FUNCTION_BLOCK FB_Observer_LWORD EXTENDS FB_AbstractObserver
VAR
    _nVal:              LWORD;
END_VAR

METHOD FB_init : BOOL
VAR_INPUT
	bInitRetains : BOOL; // if TRUE, the retain variables are initialized (warm start / cold start)
	bInCopyCode : BOOL;  // if TRUE, the instance afterwards gets moved into the copy code (online change)
END_VAR
THIS^._nTypeClass := __SYSTEM.TYPE_CLASS.TYPE_LWORD;
THIS^._pVal := ADR(THIS^._nVal);
THIS^._nSize := SIZEOF(THIS^._nVal);
END_METHOD

PROPERTY nValue64 : LWORD
GET
nValue64 := THIS^._nVal;
END_GET
END_PROPERTY

END_FUNCTION_BLOCK

(* stored: Version 1.1.0.1, ProductVersion 3.1.4024.12
   POU FB_Observer_LWORD: Id {5cea1ad3-7dae-0455-15e2-2fead871edb9}, SpecialFunc None
   Method FB_init: Id {59ef49af-99d6-06fc-1dd9-c1e7de4d5ebe}
   Property nValue64: Id {a07f065d-889f-00ee-3d6d-ec4f5f290776}
   Get Get: Id {ac783166-2029-0f31-3739-e8871e71d900} *)
